FUNCTION_BLOCK FB_ManualStrategy IMPLEMENTS I_ModeStrategy
VAR
END_VAR

METHOD GetModeName : STRING
GetModeName := 'MANUAL';
END_METHOD

METHOD Reset
END_METHOD

METHOD ShouldLoop : BOOL
ShouldLoop := FALSE;
END_METHOD

END_FUNCTION_BLOCK

(* stored: Version 1.1.0.1, ProductVersion 3.1.4024.16
   POU FB_ManualStrategy: Id {e9ae5da6-e60a-4aea-9eeb-53096ea25349}, SpecialFunc None
   Method GetModeName: Id {6792748e-2a6b-47c1-91f0-63c5b9153263}
   Method Reset: Id {63d4b590-5815-4bc0-bcaf-15c5322a6648}
   Method ShouldLoop: Id {455630bb-d218-4ae4-a308-8698edfe9371} *)
